{region '#Template'}
	{attribute 'Version' := '5.0.0.0'}
	{attribute 'Tags' := '"LCID": "1031", "Text": "General, Settings, Parameters, Basics"'}
	{attribute 'Tags' := '"LCID": "1033", "Text": "General, Settings, Parameters, Basics"'}
	{attribute 'Using' := '"Type": "Template", "URI": "BA2_Param"'}
	{attribute 'Description' := '"LCID": "1031", "Text": "Witterungsparameter für die Templates"'}
	{attribute 'Description' := '"LCID": "1033", "Text": "Weather parameters for the templates"'}
{endregion}
FUNCTION_BLOCK FB_BA_WeatherParameter EXTENDS FB_BA_View
VAR_INPUT
	fTWth					: REAL;	//	Weather temperature
END_VAR
VAR_OUTPUT
	fSpFrstProtec			: REAL;  // frost protection setpoint. for eg. Heating circutis in protection mode
	fTWthLowLimit			: REAL;  // below this value all frostprotection funcktions in HVAC-Plants will be enabled
	bTWthLowLimit			: BOOL;  // is TRUE when the outside temperature is below the value from fTWthLowLimit 
	fTWthDamped				: REAL;  // damped outside temperature
	bTWthDampedLowLimit		: BOOL;	
END_VAR
VAR_INPUT CONSTANT
	SpFrstProtec			: FB_BA_AV_Op;		
	TWthLowLimitVal			: FB_BA_AV_Op;																
	TWthLowLimit			: FB_BA_BV_Op;								
	TWthDamped				: FB_BA_AV_Op;		
	TWthDampedLowLimit		: FB_BA_BV_Op;	
END_VAR
VAR
	TWthLowLimitHys			: FB_BA_Swi2P;
	Average					: FB_BA_TiAvrg;
	TWthDampedLowLimitHys	: FB_BA_Swi2P;
END_VAR

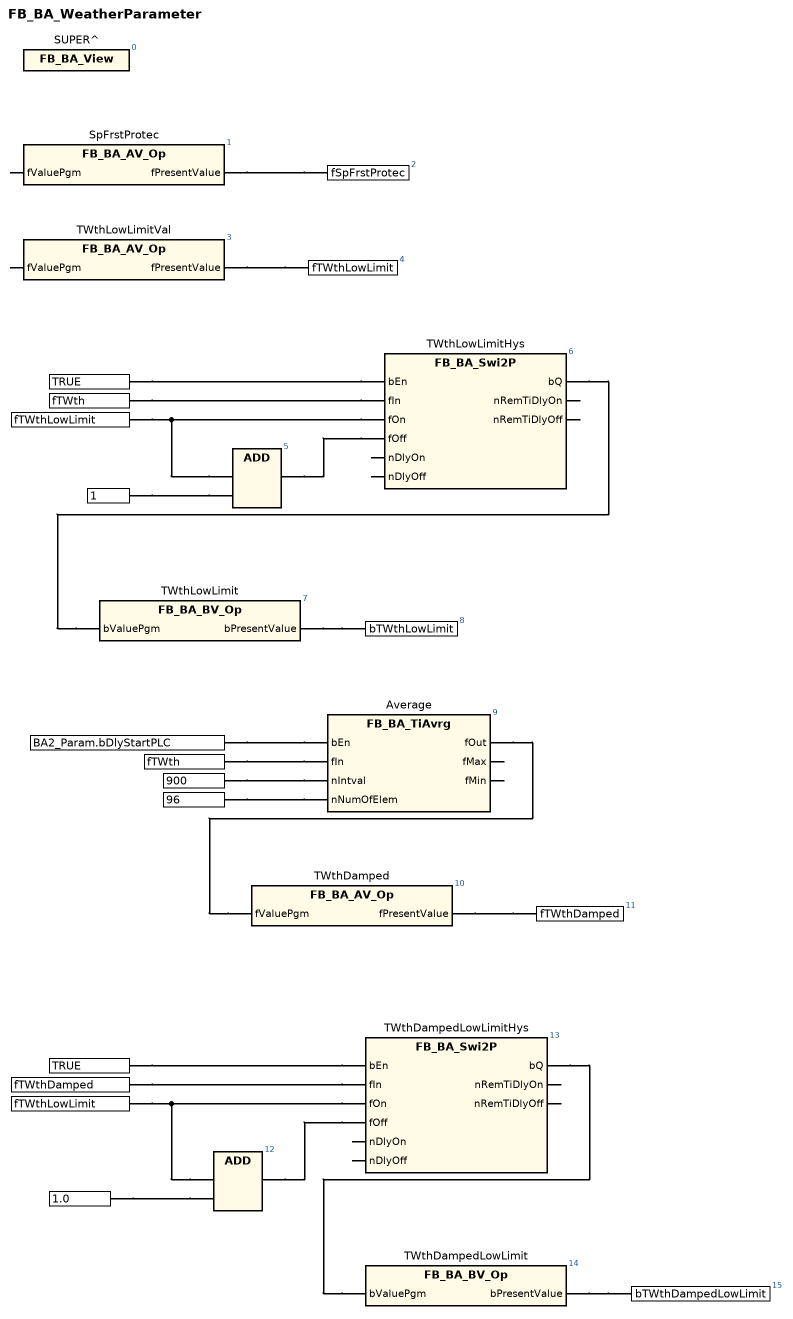
SUPER^(); // FB_BA_View
SpFrstProtec(); // FB_BA_AV_Op
fSpFrstProtec := SpFrstProtec.fPresentValue;
TWthLowLimitVal(); // FB_BA_AV_Op
fTWthLowLimit := TWthLowLimitVal.fPresentValue;
TWthLowLimitHys(bEn := TRUE, fIn := fTWth, fOn := fTWthLowLimit, fOff := fTWthLowLimit + 1); // FB_BA_Swi2P
TWthLowLimit(bValuePgm := TWthLowLimitHys.bQ); // FB_BA_BV_Op
bTWthLowLimit := TWthLowLimit.bPresentValue;
Average(bEn := BA2_Param.bDlyStartPLC, fIn := fTWth, nIntval := 900, nNumOfElem := 96); // FB_BA_TiAvrg
TWthDamped(fValuePgm := Average.fOut); // FB_BA_AV_Op
fTWthDamped := TWthDamped.fPresentValue;
TWthDampedLowLimitHys(bEn := TRUE, fIn := fTWthDamped, fOn := fTWthLowLimit, fOff := fTWthLowLimit + 1.0); // FB_BA_Swi2P
TWthDampedLowLimit(bValuePgm := TWthDampedLowLimitHys.bQ); // FB_BA_BV_Op
bTWthDampedLowLimit := TWthDampedLowLimit.bPresentValue;

METHOD FB_init : BOOL
VAR_INPUT
	bInitRetains : BOOL; // if TRUE, the retain variables are initialized (warm start / cold start)
	bInCopyCode : BOOL;  // if TRUE, the instance afterwards gets moved into the copy code (online change)
END_VAR
SpFrstProtec.iParent				:= THIS^;
SpFrstProtec.iLabel					:= LblCtl_SetpointFrostProtection;
SpFrstProtec.eUnit					:= E_BA_Unit.eTemperature_DegreesCelsius;  
SpFrstProtec.fValueRm				:= 5.0;
SpFrstProtec.fCOVIncrement			:= BA2_Param.fDefCOVIncrement;							

TWthLowLimitVal.iParent				:= THIS^;
TWthLowLimitVal.iLabel				:= LblCtl_SetpointMinimumOutsideTemperature;
TWthLowLimitVal.eUnit				:= E_BA_Unit.eTemperature_DegreesCelsius;  
TWthLowLimitVal.fValueRm			:= 8.0;
TWthLowLimitVal.fCOVIncrement		:= BA2_Param.fDefCOVIncrement;							

TWthLowLimit.iParent				:= THIS^;	
TWthLowLimit.iLabel					:= LblCtl_OperationalMessageTemperatureWeatherLowLimit;
TWthLowLimit.sInactiveText			:= txtEvent_Off;
TWthLowLimit.sActiveText			:= txtEvent_On;
TWthLowLimit.bValueRm				:= FALSE;		
TWthLowLimit.eToggleMode 			:= E_BA_ToggleMode.eSwitch;

TWthDamped.iParent					:= THIS^;
TWthDamped.iLabel					:= LblCtl_MeanDamped;
TWthDamped.eUnit					:= E_BA_Unit.eTemperature_DegreesCelsius;  
TWthDamped.fValueRm					:= 0.0;
TWthDamped.fCOVIncrement			:= BA2_Param.fDefCOVIncrement;							

TWthDampedLowLimit.iParent			:= THIS^;	
TWthDampedLowLimit.iLabel			:= LblCtl_OperationalMessageTemperatureWeatherDampedLowLimit;	
TWthDampedLowLimit.sInactiveText	:= txtEvent_Off;
TWthDampedLowLimit.sActiveText		:= txtEvent_On;
TWthDampedLowLimit.bValueRm			:= FALSE;								
TWthDampedLowLimit.eToggleMode 		:= E_BA_ToggleMode.eSwitch;
END_METHOD

END_FUNCTION_BLOCK

(* stored: Version 1.1.0.1, ProductVersion 3.1.4024.12
   POU FB_BA_WeatherParameter: Id {8b415902-969b-4347-97ae-4acd943bf041}, SpecialFunc None
   Method FB_init: Id {3af963c5-9735-4a2b-8918-ad6bee54a2a8} *)
